// Mitsubishi GX Works2 project: 탁상 타이머 토익스피킹 시계0912   PLC: Q03UDV

PROGRAM MAIN
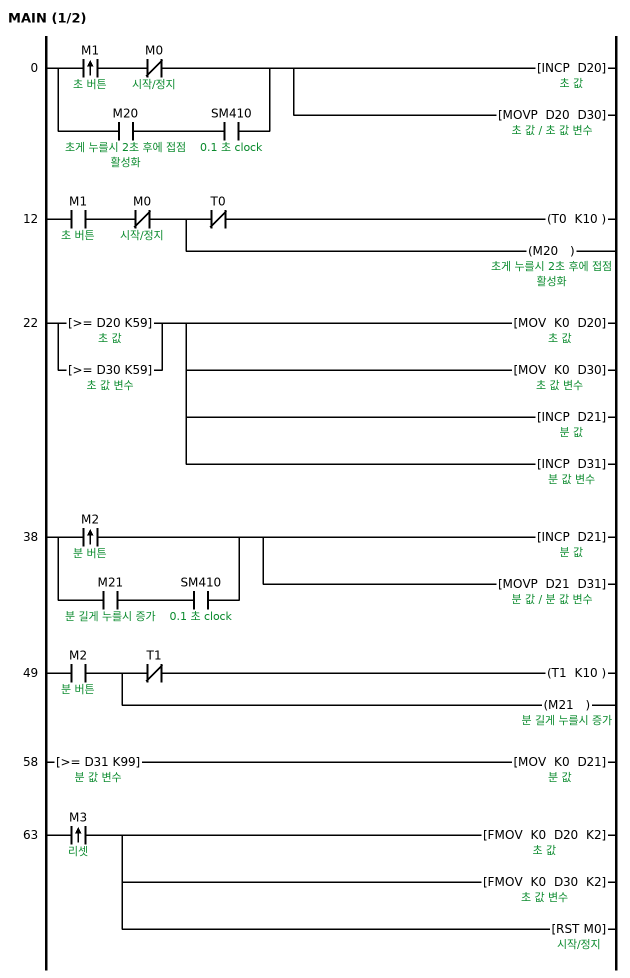
0     LDP     M1  ; 초 버튼
      ANI     M0  ; 시작/정지
      LD      M20  ; 초게 누를시 2초 후에 접점 활성화
      AND     SM410  ; 0.1 초 clock
      ORB
      INCP    D20  ; 초 값
      MOVP    D20 D30  ; 초 값 변수
12    LD      M1  ; 초 버튼
      ANI     M0  ; 시작/정지
      MPS
      ANI     T0
      OUT     T0 K10
      MPP
      OUT     M20  ; 초게 누를시 2초 후에 접점 활성화
22    LD>=    D20 K59  ; 초 값
      OR>=    D30 K59  ; 초 값 변수
      MOV     K0 D20
      MOV     K0 D30
      INCP    D21  ; 분 값
      INCP    D31  ; 분 값 변수
38    LDP     M2  ; 분 버튼
      LD      M21  ; 분 길게 누를시 증가
      AND     SM410  ; 0.1 초 clock
      ORB
      INCP    D21
      MOVP    D21 D31
49    LD      M2  ; 분 버튼
      MPS
      ANI     T1
      OUT     T1 K10
      MPP
      OUT     M21  ; 분 길게 누를시 증가
58    LD>=    D31 K99  ; 분 값 변수
      MOV     K0 D21
63    LDP     M3  ; 리셋
      FMOV    K0 D20 K2
      FMOV    K0 D30 K2
      RST     M0  ; 시작/정지
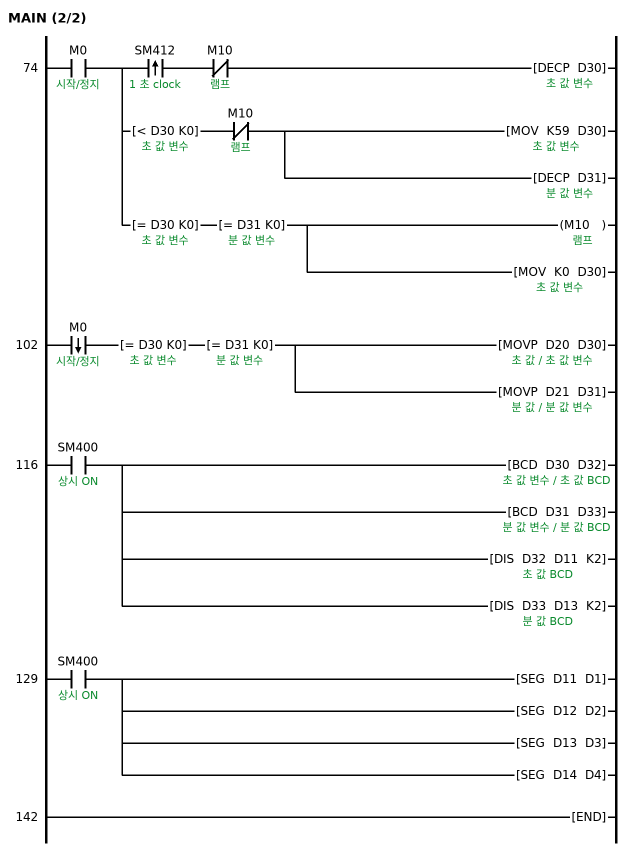
74    LD      M0  ; 시작/정지
      MPS
      ANDP    SM412  ; 1 초 clock
      ANI     M10  ; 램프
      DECP    D30
      MRD
      AND<    D30 K0  ; 초 값 변수
      ANI     M10  ; 램프
      MOV     K59 D30
      DECP    D31
      MPP
      AND=    D30 K0  ; 초 값 변수
      AND=    D31 K0  ; 분 값 변수
      OUT     M10  ; 램프
      MOV     K0 D30
102   LDF     M0  ; 시작/정지
      AND=    D30 K0  ; 초 값 변수
      AND=    D31 K0  ; 분 값 변수
      MOVP    D20 D30
      MOVP    D21 D31
116   LD      SM400  ; 상시 ON
      BCD     D30 D32  ; 초 값 BCD
      BCD     D31 D33  ; 분 값 BCD
      DIS     D32 D11 K2
      DIS     D33 D13 K2
129   LD      SM400  ; 상시 ON
      SEG     D11 D1
      SEG     D12 D2
      SEG     D13 D3
      SEG     D14 D4
142   END
END_PROGRAM
